// TIA Portal V21 export
FUNCTION "PidInitialisation" : Void   // FC3, LAD
{ S7_Optimized_Access := 'TRUE' }
// stored: SetENOAutomatically false
BEGIN

REGION Network 2: CV30 Parameters SIP
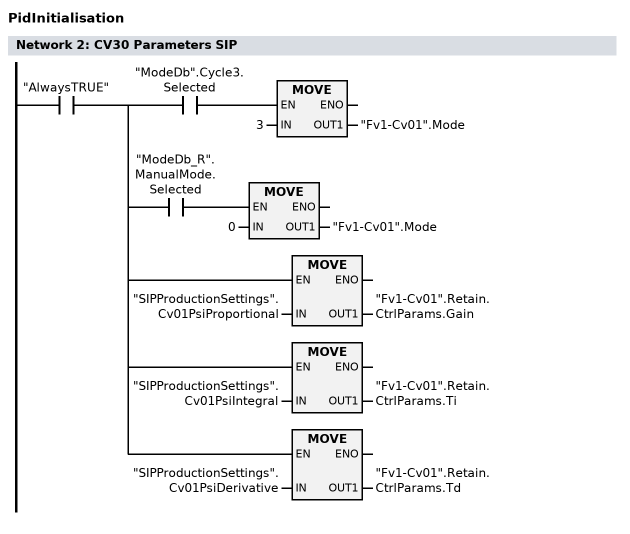
   RUNG wire#powerrail
      Contact( "AlwaysTRUE" )
      wire#w1
      Contact( "ModeDb".Cycle3.Selected )
      { S7_GenerateENO := "TRUE" } Move(in := 3, out1 => "Fv1-Cv01".Mode)
   END_RUNG
   RUNG wire#w1
      Contact( "ModeDb_R".ManualMode.Selected )
      { S7_GenerateENO := "TRUE" } Move(in := 0, out1 => "Fv1-Cv01".Mode)
   END_RUNG
   RUNG wire#w1
      { S7_GenerateENO := "TRUE" } Move(in := "SIPProductionSettings".Cv01PsiProportional, out1 => "Fv1-Cv01".Retain.CtrlParams.Gain)
   END_RUNG
   RUNG wire#w1
      { S7_GenerateENO := "TRUE" } Move(in := "SIPProductionSettings".Cv01PsiIntegral, out1 => "Fv1-Cv01".Retain.CtrlParams.Ti)
   END_RUNG
   RUNG wire#w1
      { S7_GenerateENO := "TRUE" } Move(in := "SIPProductionSettings".Cv01PsiDerivative, out1 => "Fv1-Cv01".Retain.CtrlParams.Td)
   END_RUNG
   // the same network as SCL:
   IF "AlwaysTRUE" AND "ModeDb".Cycle3.Selected THEN "Fv1-Cv01".Mode := 3; END_IF;
   IF "AlwaysTRUE" AND "ModeDb_R".ManualMode.Selected THEN "Fv1-Cv01".Mode := 0; END_IF;
   IF "AlwaysTRUE" THEN
       "Fv1-Cv01".Retain.CtrlParams.Gain := "SIPProductionSettings".Cv01PsiProportional;
       "Fv1-Cv01".Retain.CtrlParams.Ti := "SIPProductionSettings".Cv01PsiIntegral;
       "Fv1-Cv01".Retain.CtrlParams.Td := "SIPProductionSettings".Cv01PsiDerivative;
   END_IF;
END_REGION
END_FUNCTION
